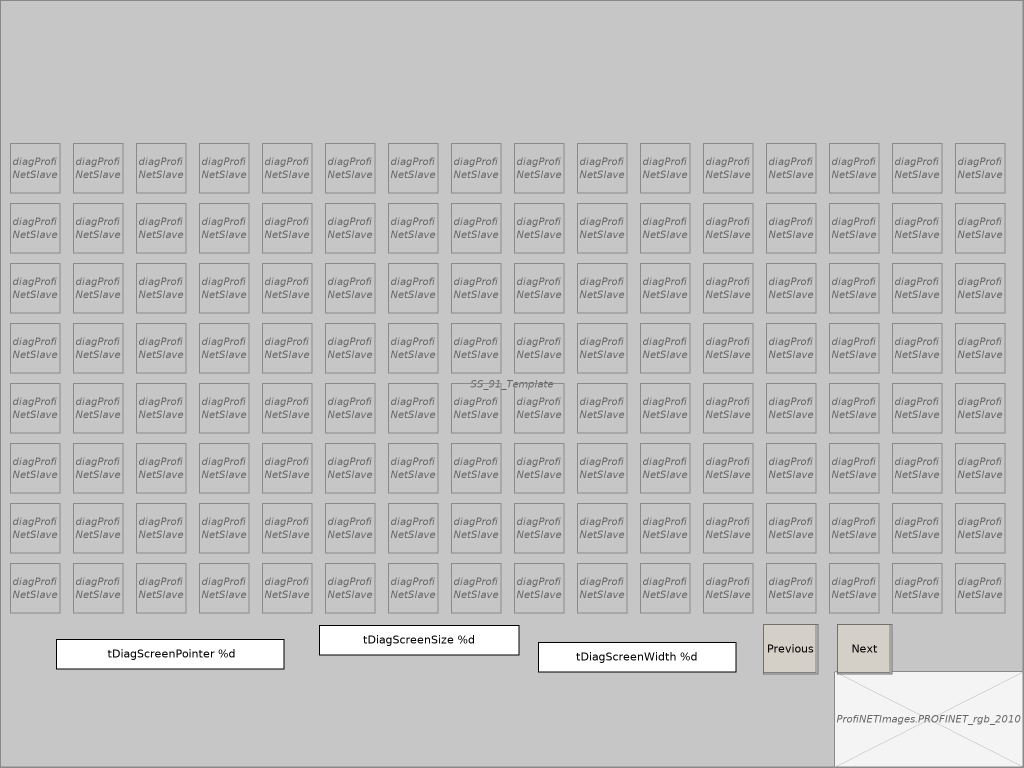
VISUALIZATION DI_03_ProfiNet  // 1024x768
    Frame (0,0 1024x768)
        shows SS_91_Template(header := HMIData.hmiHeader)
    Frame (10,143 50x50)
        shows diagProfiNetSlave(dataValues := ProfiNetDiag.diagScreen[1])
    Frame (73,143 50x50)
        shows diagProfiNetSlave(dataValues := ProfiNetDiag.diagScreen[2])
    Frame (136,143 50x50)
        shows diagProfiNetSlave(dataValues := ProfiNetDiag.diagScreen[3])
    Frame (199,143 50x50)
        shows diagProfiNetSlave(dataValues := ProfiNetDiag.diagScreen[4])
    Frame (262,143 50x50)
        shows diagProfiNetSlave(dataValues := ProfiNetDiag.diagScreen[5])
    Frame (325,143 50x50)
        shows diagProfiNetSlave(dataValues := ProfiNetDiag.diagScreen[6])
    Frame (388,143 50x50)
        shows diagProfiNetSlave(dataValues := ProfiNetDiag.diagScreen[7])
    Frame (451,143 50x50)
        shows diagProfiNetSlave(dataValues := ProfiNetDiag.diagScreen[8])
    Frame (514,143 50x50)
        shows diagProfiNetSlave(dataValues := ProfiNetDiag.diagScreen[9])
    Frame (577,143 50x50)
        shows diagProfiNetSlave(dataValues := ProfiNetDiag.diagScreen[10])
    Frame (640,143 50x50)
        shows diagProfiNetSlave(dataValues := ProfiNetDiag.diagScreen[11])
    Frame (703,143 50x50)
        shows diagProfiNetSlave(dataValues := ProfiNetDiag.diagScreen[12])
    Frame (766,143 50x50)
        shows diagProfiNetSlave(dataValues := ProfiNetDiag.diagScreen[13])
    Frame (829,143 50x50)
        shows diagProfiNetSlave(dataValues := ProfiNetDiag.diagScreen[14])
    Frame (892,143 50x50)
        shows diagProfiNetSlave(dataValues := ProfiNetDiag.diagScreen[15])
    Frame (955,143 50x50)
        shows diagProfiNetSlave(dataValues := ProfiNetDiag.diagScreen[16])
    Image (834,671 190x96), image: ProfiNETImages.PROFINET_rgb_2010
    Button (763,624 55x50), "Previous"
        tap ProfiNetDiag.btnPrevious
    Button (837,624 55x50), "Next"
        tap ProfiNetDiag.btnNext
    Rectangle (56,639 228x30), "tDiagScreenPointer %d", text variable: pouPROFINETdiag.tDiagScreenPointer
    Rectangle (319,625 200x30), "tDiagScreenSize %d", text variable: pouPROFINETdiag.tDiagScreenSize
    Rectangle (538,642 198x30), "tDiagScreenWidth %d", text variable: pouPROFINETdiag.tDiagScreenWidth
    Frame (10,203 50x50)
        shows diagProfiNetSlave(dataValues := ProfiNetDiag.diagScreen[1])
    Frame (73,203 50x50)
        shows diagProfiNetSlave(dataValues := ProfiNetDiag.diagScreen[2])
    Frame (136,203 50x50)
        shows diagProfiNetSlave(dataValues := ProfiNetDiag.diagScreen[3])
    Frame (199,203 50x50)
        shows diagProfiNetSlave(dataValues := ProfiNetDiag.diagScreen[4])
    Frame (262,203 50x50)
        shows diagProfiNetSlave(dataValues := ProfiNetDiag.diagScreen[5])
    Frame (325,203 50x50)
        shows diagProfiNetSlave(dataValues := ProfiNetDiag.diagScreen[6])
    Frame (388,203 50x50)
        shows diagProfiNetSlave(dataValues := ProfiNetDiag.diagScreen[7])
    Frame (451,203 50x50)
        shows diagProfiNetSlave(dataValues := ProfiNetDiag.diagScreen[8])
    Frame (514,203 50x50)
        shows diagProfiNetSlave(dataValues := ProfiNetDiag.diagScreen[9])
    Frame (577,203 50x50)
        shows diagProfiNetSlave(dataValues := ProfiNetDiag.diagScreen[10])
    Frame (640,203 50x50)
        shows diagProfiNetSlave(dataValues := ProfiNetDiag.diagScreen[11])
    Frame (703,203 50x50)
        shows diagProfiNetSlave(dataValues := ProfiNetDiag.diagScreen[12])
    Frame (766,203 50x50)
        shows diagProfiNetSlave(dataValues := ProfiNetDiag.diagScreen[13])
    Frame (829,203 50x50)
        shows diagProfiNetSlave(dataValues := ProfiNetDiag.diagScreen[14])
    Frame (892,203 50x50)
        shows diagProfiNetSlave(dataValues := ProfiNetDiag.diagScreen[15])
    Frame (955,203 50x50)
        shows diagProfiNetSlave(dataValues := ProfiNetDiag.diagScreen[16])
    Frame (10,263 50x50)
        shows diagProfiNetSlave(dataValues := ProfiNetDiag.diagScreen[1])
    Frame (73,263 50x50)
        shows diagProfiNetSlave(dataValues := ProfiNetDiag.diagScreen[2])
    Frame (136,263 50x50)
        shows diagProfiNetSlave(dataValues := ProfiNetDiag.diagScreen[3])
    Frame (199,263 50x50)
        shows diagProfiNetSlave(dataValues := ProfiNetDiag.diagScreen[4])
    Frame (262,263 50x50)
        shows diagProfiNetSlave(dataValues := ProfiNetDiag.diagScreen[5])
    Frame (325,263 50x50)
        shows diagProfiNetSlave(dataValues := ProfiNetDiag.diagScreen[6])
    Frame (388,263 50x50)
        shows diagProfiNetSlave(dataValues := ProfiNetDiag.diagScreen[7])
    Frame (451,263 50x50)
        shows diagProfiNetSlave(dataValues := ProfiNetDiag.diagScreen[8])
    Frame (514,263 50x50)
        shows diagProfiNetSlave(dataValues := ProfiNetDiag.diagScreen[9])
    Frame (577,263 50x50)
        shows diagProfiNetSlave(dataValues := ProfiNetDiag.diagScreen[10])
    Frame (640,263 50x50)
        shows diagProfiNetSlave(dataValues := ProfiNetDiag.diagScreen[11])
    Frame (703,263 50x50)
        shows diagProfiNetSlave(dataValues := ProfiNetDiag.diagScreen[12])
    Frame (766,263 50x50)
        shows diagProfiNetSlave(dataValues := ProfiNetDiag.diagScreen[13])
    Frame (829,263 50x50)
        shows diagProfiNetSlave(dataValues := ProfiNetDiag.diagScreen[14])
    Frame (892,263 50x50)
        shows diagProfiNetSlave(dataValues := ProfiNetDiag.diagScreen[15])
    Frame (955,263 50x50)
        shows diagProfiNetSlave(dataValues := ProfiNetDiag.diagScreen[16])
    Frame (10,323 50x50)
        shows diagProfiNetSlave(dataValues := ProfiNetDiag.diagScreen[1])
    Frame (73,323 50x50)
        shows diagProfiNetSlave(dataValues := ProfiNetDiag.diagScreen[2])
    Frame (136,323 50x50)
        shows diagProfiNetSlave(dataValues := ProfiNetDiag.diagScreen[3])
    Frame (199,323 50x50)
        shows diagProfiNetSlave(dataValues := ProfiNetDiag.diagScreen[4])
    Frame (262,323 50x50)
        shows diagProfiNetSlave(dataValues := ProfiNetDiag.diagScreen[5])
    Frame (325,323 50x50)
        shows diagProfiNetSlave(dataValues := ProfiNetDiag.diagScreen[6])
    Frame (388,323 50x50)
        shows diagProfiNetSlave(dataValues := ProfiNetDiag.diagScreen[7])
    Frame (451,323 50x50)
        shows diagProfiNetSlave(dataValues := ProfiNetDiag.diagScreen[8])
    Frame (514,323 50x50)
        shows diagProfiNetSlave(dataValues := ProfiNetDiag.diagScreen[9])
    Frame (577,323 50x50)
        shows diagProfiNetSlave(dataValues := ProfiNetDiag.diagScreen[10])
    Frame (640,323 50x50)
        shows diagProfiNetSlave(dataValues := ProfiNetDiag.diagScreen[11])
    Frame (703,323 50x50)
        shows diagProfiNetSlave(dataValues := ProfiNetDiag.diagScreen[12])
    Frame (766,323 50x50)
        shows diagProfiNetSlave(dataValues := ProfiNetDiag.diagScreen[13])
    Frame (829,323 50x50)
        shows diagProfiNetSlave(dataValues := ProfiNetDiag.diagScreen[14])
    Frame (892,323 50x50)
        shows diagProfiNetSlave(dataValues := ProfiNetDiag.diagScreen[15])
    Frame (955,323 50x50)
        shows diagProfiNetSlave(dataValues := ProfiNetDiag.diagScreen[16])
    Frame (10,383 50x50)
        shows diagProfiNetSlave(dataValues := ProfiNetDiag.diagScreen[1])
    Frame (73,383 50x50)
        shows diagProfiNetSlave(dataValues := ProfiNetDiag.diagScreen[2])
    Frame (136,383 50x50)
        shows diagProfiNetSlave(dataValues := ProfiNetDiag.diagScreen[3])
    Frame (199,383 50x50)
        shows diagProfiNetSlave(dataValues := ProfiNetDiag.diagScreen[4])
    Frame (262,383 50x50)
        shows diagProfiNetSlave(dataValues := ProfiNetDiag.diagScreen[5])
    Frame (325,383 50x50)
        shows diagProfiNetSlave(dataValues := ProfiNetDiag.diagScreen[6])
    Frame (388,383 50x50)
        shows diagProfiNetSlave(dataValues := ProfiNetDiag.diagScreen[7])
    Frame (451,383 50x50)
        shows diagProfiNetSlave(dataValues := ProfiNetDiag.diagScreen[8])
    Frame (514,383 50x50)
        shows diagProfiNetSlave(dataValues := ProfiNetDiag.diagScreen[9])
    Frame (577,383 50x50)
        shows diagProfiNetSlave(dataValues := ProfiNetDiag.diagScreen[10])
    Frame (640,383 50x50)
        shows diagProfiNetSlave(dataValues := ProfiNetDiag.diagScreen[11])
    Frame (703,383 50x50)
        shows diagProfiNetSlave(dataValues := ProfiNetDiag.diagScreen[12])
    Frame (766,383 50x50)
        shows diagProfiNetSlave(dataValues := ProfiNetDiag.diagScreen[13])
    Frame (829,383 50x50)
        shows diagProfiNetSlave(dataValues := ProfiNetDiag.diagScreen[14])
    Frame (892,383 50x50)
        shows diagProfiNetSlave(dataValues := ProfiNetDiag.diagScreen[15])
    Frame (955,383 50x50)
        shows diagProfiNetSlave(dataValues := ProfiNetDiag.diagScreen[16])
    Frame (10,443 50x50)
        shows diagProfiNetSlave(dataValues := ProfiNetDiag.diagScreen[1])
    Frame (73,443 50x50)
        shows diagProfiNetSlave(dataValues := ProfiNetDiag.diagScreen[2])
    Frame (136,443 50x50)
        shows diagProfiNetSlave(dataValues := ProfiNetDiag.diagScreen[3])
    Frame (199,443 50x50)
        shows diagProfiNetSlave(dataValues := ProfiNetDiag.diagScreen[4])
    Frame (262,443 50x50)
        shows diagProfiNetSlave(dataValues := ProfiNetDiag.diagScreen[5])
    Frame (325,443 50x50)
        shows diagProfiNetSlave(dataValues := ProfiNetDiag.diagScreen[6])
    Frame (388,443 50x50)
        shows diagProfiNetSlave(dataValues := ProfiNetDiag.diagScreen[7])
    Frame (451,443 50x50)
        shows diagProfiNetSlave(dataValues := ProfiNetDiag.diagScreen[8])
    Frame (514,443 50x50)
        shows diagProfiNetSlave(dataValues := ProfiNetDiag.diagScreen[9])
    Frame (577,443 50x50)
        shows diagProfiNetSlave(dataValues := ProfiNetDiag.diagScreen[10])
    Frame (640,443 50x50)
        shows diagProfiNetSlave(dataValues := ProfiNetDiag.diagScreen[11])
    Frame (703,443 50x50)
        shows diagProfiNetSlave(dataValues := ProfiNetDiag.diagScreen[12])
    Frame (766,443 50x50)
        shows diagProfiNetSlave(dataValues := ProfiNetDiag.diagScreen[13])
    Frame (829,443 50x50)
        shows diagProfiNetSlave(dataValues := ProfiNetDiag.diagScreen[14])
    Frame (892,443 50x50)
        shows diagProfiNetSlave(dataValues := ProfiNetDiag.diagScreen[15])
    Frame (955,443 50x50)
        shows diagProfiNetSlave(dataValues := ProfiNetDiag.diagScreen[16])
    Frame (10,503 50x50)
        shows diagProfiNetSlave(dataValues := ProfiNetDiag.diagScreen[1])
    Frame (73,503 50x50)
        shows diagProfiNetSlave(dataValues := ProfiNetDiag.diagScreen[2])
    Frame (136,503 50x50)
        shows diagProfiNetSlave(dataValues := ProfiNetDiag.diagScreen[3])
    Frame (199,503 50x50)
        shows diagProfiNetSlave(dataValues := ProfiNetDiag.diagScreen[4])
    Frame (262,503 50x50)
        shows diagProfiNetSlave(dataValues := ProfiNetDiag.diagScreen[5])
    Frame (325,503 50x50)
        shows diagProfiNetSlave(dataValues := ProfiNetDiag.diagScreen[6])
    Frame (388,503 50x50)
        shows diagProfiNetSlave(dataValues := ProfiNetDiag.diagScreen[7])
    Frame (451,503 50x50)
        shows diagProfiNetSlave(dataValues := ProfiNetDiag.diagScreen[8])
    Frame (514,503 50x50)
        shows diagProfiNetSlave(dataValues := ProfiNetDiag.diagScreen[9])
    Frame (577,503 50x50)
        shows diagProfiNetSlave(dataValues := ProfiNetDiag.diagScreen[10])
    Frame (640,503 50x50)
        shows diagProfiNetSlave(dataValues := ProfiNetDiag.diagScreen[11])
    Frame (703,503 50x50)
        shows diagProfiNetSlave(dataValues := ProfiNetDiag.diagScreen[12])
    Frame (766,503 50x50)
        shows diagProfiNetSlave(dataValues := ProfiNetDiag.diagScreen[13])
    Frame (829,503 50x50)
        shows diagProfiNetSlave(dataValues := ProfiNetDiag.diagScreen[14])
    Frame (892,503 50x50)
        shows diagProfiNetSlave(dataValues := ProfiNetDiag.diagScreen[15])
    Frame (955,503 50x50)
        shows diagProfiNetSlave(dataValues := ProfiNetDiag.diagScreen[16])
    Frame (10,563 50x50)
        shows diagProfiNetSlave(dataValues := ProfiNetDiag.diagScreen[1])
    Frame (73,563 50x50)
        shows diagProfiNetSlave(dataValues := ProfiNetDiag.diagScreen[2])
    Frame (136,563 50x50)
        shows diagProfiNetSlave(dataValues := ProfiNetDiag.diagScreen[3])
    Frame (199,563 50x50)
        shows diagProfiNetSlave(dataValues := ProfiNetDiag.diagScreen[4])
    Frame (262,563 50x50)
        shows diagProfiNetSlave(dataValues := ProfiNetDiag.diagScreen[5])
    Frame (325,563 50x50)
        shows diagProfiNetSlave(dataValues := ProfiNetDiag.diagScreen[6])
    Frame (388,563 50x50)
        shows diagProfiNetSlave(dataValues := ProfiNetDiag.diagScreen[7])
    Frame (451,563 50x50)
        shows diagProfiNetSlave(dataValues := ProfiNetDiag.diagScreen[8])
    Frame (514,563 50x50)
        shows diagProfiNetSlave(dataValues := ProfiNetDiag.diagScreen[9])
    Frame (577,563 50x50)
        shows diagProfiNetSlave(dataValues := ProfiNetDiag.diagScreen[10])
    Frame (640,563 50x50)
        shows diagProfiNetSlave(dataValues := ProfiNetDiag.diagScreen[11])
    Frame (703,563 50x50)
        shows diagProfiNetSlave(dataValues := ProfiNetDiag.diagScreen[12])
    Frame (766,563 50x50)
        shows diagProfiNetSlave(dataValues := ProfiNetDiag.diagScreen[13])
    Frame (829,563 50x50)
        shows diagProfiNetSlave(dataValues := ProfiNetDiag.diagScreen[14])
    Frame (892,563 50x50)
        shows diagProfiNetSlave(dataValues := ProfiNetDiag.diagScreen[15])
    Frame (955,563 50x50)
        shows diagProfiNetSlave(dataValues := ProfiNetDiag.diagScreen[16])
END_VISUALIZATION

(* stored: Version 1.1.0.1, ProductVersion 3.1.4024.12
   Visu DI_03_ProfiNet: Id {12fd3784-54bb-476d-9c00-b84e219884e2} *)
